(* CODESYS project Simulation_Arm_ROS2_COD_OOP.project

Project tree, tasks and I/O mapping:
  Device : CODESYS Virtual Control for Linux SL, CODESYS, order no. 2302000005, version 4.22.0.0
    application Application
      libraries: Standard, 3.5.22.0 (System); VisuDialogs, * (System)
      task MainTask (cyclic, interval t#20ms, priority 1) calls PLC_PRG, PRG_Visu [Visualisierung]
      program PLC_PRG [ST]
      Kommunikationsverwalter
        OPC UA Server
          Symbolgruppe
      global variables GVL_OPCUA
      visualisation Topics_Vis
      program PRG_VISU [ST]
      Structs/
        ST_RobotStatus/
          data type ST_RobotStatus
          data type ST_Pose_Axis
          data type ST_Pose_TCP
          data type ST_Modes
        ST_RobotAction/
          data type RobotAction
        ST_RobotCommand/
          data type RobotCommand
          data type ST_Servo_Axis
          data type ST_Servo_TCP
      old_code/
        data type Manuell_Achse
        data type TCP_Pose
        data type JointState
        FB_Robot/
          function block FB_Robot [FBD]
          function block FB_Watchdog [ST]
          function block FB_RobotCommand [ST]
      Interfaces/
        interface IF_RobotStatus: Ist_Pose_Axis, Ist_Pose_TCP, Ist_Mode, Client_Connection_Status, Update_Watchdog
        interface IF_RobotCommand: Soll_Pose_Axis, Soll_Pose_TCP
      function block FB_Roboter [FBD]: Update_Watchdog, Soll_Pose_Axis, Soll_Pose_TCP, Client_Connection_Status, Ist_Mode, Ist_Pose_Axis, Ist_Pose_TCP
  libraries: SM3_Robotics, * (CODESYS); VisuSymbols, 4.5.0.0 (System)
  text list GlobalTextList
*)

// Device/Application/old_code/Manuell_Achse
TYPE Manuell_Achse :
STRUCT
	axis_0_plus : BOOL;
	axis_0_minus : BOOL;
	axis_1_plus : BOOL;
	axis_1_minus : BOOL;
	axis_2_plus : BOOL;
	axis_2_minus : BOOL;
	axis_3_plus : BOOL;
	axis_3_minus : BOOL;
	axis_4_plus : BOOL;
	axis_4_minus : BOOL;
	axis_5_plus : BOOL;
	axis_5_minus : BOOL;
	//velocity_spee  einstellen
	//start manuell
END_STRUCT
END_TYPE

// Device/Application/old_code/TCP_Pose
TYPE TCP_Pose :
STRUCT
	trans_x : LREAL;
	trans_y : LREAL;
	trans_z : LREAL;
	rot_x : LREAL;
	rot_y : LREAL;
	rot_z : LREAL;
	rot_w : LREAL;
END_STRUCT
END_TYPE

//TCP Pose in kartesischen Koordinaten
//Rotation wird in quaternions uebermittelt, muss noch umgerechnet werden

// Device/Application/old_code/JointState
TYPE JointState :
STRUCT
	name :ARRAY[0..5] OF STRING;
	position :ARRAY[0..5] OF LREAL; 
	effort :ARRAY[0..5] OF LREAL;
	velocity :ARRAY[0..5] OF LREAL;
END_STRUCT
END_TYPE

// Device/Application/Structs/ST_RobotStatus/ST_RobotStatus
// Gibt den aktuellen Status des Roboters an
TYPE ST_RobotStatus :
STRUCT
	Client_Connected : BOOL;
	Watchdog_Client : INT;		// Überprüft serverseitige client verbindung
	Mode : ST_Modes;			//gibt an ob im Mode Command, Action oder idle
	Pos_Axis : ST_Pose_Axis; 	//gibt aktuelle Achspositionen an
	Pos_TCP : ST_Pose_TCP;		//gibt aktuelle tcp positionen an 
END_STRUCT
END_TYPE

// Device/Application/Structs/ST_RobotCommand/RobotCommand
TYPE RobotCommand :
STRUCT
	Client_connected: BOOL;
	Watchdog_Client: INT;
	axis_servo : ST_Servo_Axis;
	tcp_servo : ST_Servo_TCP;
END_STRUCT
END_TYPE

// Device/Application/Structs/ST_RobotAction/RobotAction
TYPE RobotAction :
STRUCT
END_STRUCT
END_TYPE

// Device/Application/Structs/ST_RobotStatus/ST_Pose_Axis
TYPE ST_Pose_Axis :
STRUCT
	axis_0 : LREAL;
	axis_1 : LREAL;
	axis_2 : LREAL;
	axis_3 : LREAL;
	axis_4 : LREAL;
	axis_5 : LREAL;
END_STRUCT
END_TYPE

// Device/Application/Structs/ST_RobotStatus/ST_Pose_TCP
TYPE ST_Pose_TCP :
STRUCT
	trans_x : LREAL;
	trans_y :  LREAL;
	trans_z : LREAL;
	rot_x : LREAL;
	rot_y : LREAL;
	rot_z : LREAL;
	rot_w : LREAL;
END_STRUCT
END_TYPE

// Device/Application/Structs/ST_RobotStatus/ST_Modes
TYPE ST_Modes :
STRUCT
	idle : BOOL;	//Ruhezustand
	command : BOOL;	//manuell
	aut : BOOL; 	//move_action
END_STRUCT
END_TYPE

// Device/Application/Structs/ST_RobotCommand/ST_Servo_Axis
TYPE ST_Servo_Axis :
STRUCT
	velocity : LREAL;	
	axis_0 : LREAL;
	axis_1 : LREAL;
	axis_2 : LREAL;
	axis_3 : LREAL;
	axis_4 : LREAL;
	axis_5 : LREAL;
END_STRUCT
END_TYPE

// Device/Application/Structs/ST_RobotCommand/ST_Servo_TCP
TYPE ST_Servo_TCP :
STRUCT
	velocity : LREAL;
	trans_x : LREAL;
	trans_y : LREAL;
	trans_z : LREAL;
	rot_x : LREAL;
	rot_y : LREAL;
	rot_z : LREAL;
	rot_w : LREAL;
END_STRUCT
END_TYPE

// Device/Application/GVL_OPCUA
{attribute 'qualified_only'}
VAR_GLOBAL
	PI : REAL := 3.14159;

	//Simulation Arm
	
	//ROS2 -> Codesys
	//topic_name_ros2 : STRUCT
	//joint_states : JointState;	
	//tcp_pose: TCP_Pose;
	
	//achse manuell verfahren
	//axis_manual : Manuell_Achse;
	


END_VAR

// Device/Application/PLC_PRG
PROGRAM PLC_PRG
VAR
END_VAR

END_PROGRAM

// Device/Application/PRG_VISU
PROGRAM PRG_Visu
VAR
    //arrStruct: ARRAY[0..6] OF LREAL;
	Robot : FB_Roboter;
	
END_VAR

Robot();

END_PROGRAM

// Device/Application/FB_Roboter
FUNCTION_BLOCK FB_Roboter IMPLEMENTS IF_RobotCommand, IF_RobotStatus
VAR_INPUT
END_VAR
VAR_OUTPUT
END_VAR
VAR
	// --- Command Variablen ---
    _soll_pose_axis : ST_Servo_Axis; // (Passend zu deinem Struct-Namen)
    _soll_pose_tcp  : ST_Servo_TCP;
    
    // --- Status Variablen ---
    _client_connection_status : BOOL;
    _ist_mode         : ST_Modes;
    _ist_pose_axis    : ST_Pose_Axis;
    _ist_pose_tcp     : ST_Pose_TCP;
END_VAR

// NETWORK 1

{warning 'Methodenimplementierung hinzufügen'}
METHOD Update_Watchdog : BOOL
END_METHOD

{attribute 'monitoring' := 'variable'}
PROPERTY Soll_Pose_Axis : ST_Servo_Axis
GET
END_GET
SET
END_SET
END_PROPERTY

{attribute 'monitoring' := 'variable'}
PROPERTY Soll_Pose_TCP : ST_Servo_TCP
GET
END_GET
SET
END_SET
END_PROPERTY

{attribute 'monitoring' := 'variable'}
PROPERTY Client_Connection_Status : BOOL
GET
Client_Connection_Status := _client_connection_status;
END_GET
SET
_client_connection_status := Client_Connection_Status;
END_SET
END_PROPERTY

{attribute 'monitoring' := 'variable'}
PROPERTY Ist_Mode : ST_Modes
GET
Ist_Mode := _ist_mode;
END_GET
SET
_ist_mode := Ist_Mode;
END_SET
END_PROPERTY

{attribute 'monitoring' := 'variable'}
PROPERTY Ist_Pose_Axis : ST_Pose_Axis
GET
Ist_Pose_Axis := _ist_pose_axis;
END_GET
SET
_ist_pose_axis := Ist_Pose_Axis;
END_SET
END_PROPERTY

{attribute 'monitoring' := 'variable'}
PROPERTY Ist_Pose_TCP : ST_Pose_TCP
GET
Ist_Pose_TCP := _ist_pose_tcp;
END_GET
SET
_ist_pose_tcp := Ist_Pose_TCP;
END_SET
END_PROPERTY

END_FUNCTION_BLOCK

// Device/Application/Interfaces/IF_RobotCommand
INTERFACE IF_RobotCommand

PROPERTY Soll_Pose_Axis : ST_Servo_Axis
SET
END_SET
GET
END_GET
END_PROPERTY

PROPERTY Soll_Pose_TCP : ST_Servo_TCP
SET
END_SET
GET
END_GET
END_PROPERTY

END_INTERFACE

// Device/Application/Interfaces/IF_RobotStatus
INTERFACE IF_RobotStatus

PROPERTY Ist_Pose_Axis : ST_Pose_Axis
GET
END_GET
END_PROPERTY

PROPERTY Ist_Pose_TCP : ST_Pose_TCP
GET
END_GET
END_PROPERTY

PROPERTY Ist_Mode : ST_Modes
SET
END_SET
GET
END_GET
END_PROPERTY

PROPERTY Client_Connection_Status : BOOL
SET
END_SET
GET
END_GET
END_PROPERTY

METHOD Update_Watchdog : BOOL
VAR_INPUT
END_VAR
END_METHOD

END_INTERFACE

// Device/Application/old_code/FB_Robot/FB_Robot
FUNCTION_BLOCK FB_Robot
VAR_INPUT
	Command: RobotCommand;
END_VAR
VAR_OUTPUT
	Status: ST_RobotStatus;
END_VAR
VAR
	robotcommand : FB_RobotCommand;
	Watchdog: FB_Watchdog;
END_VAR

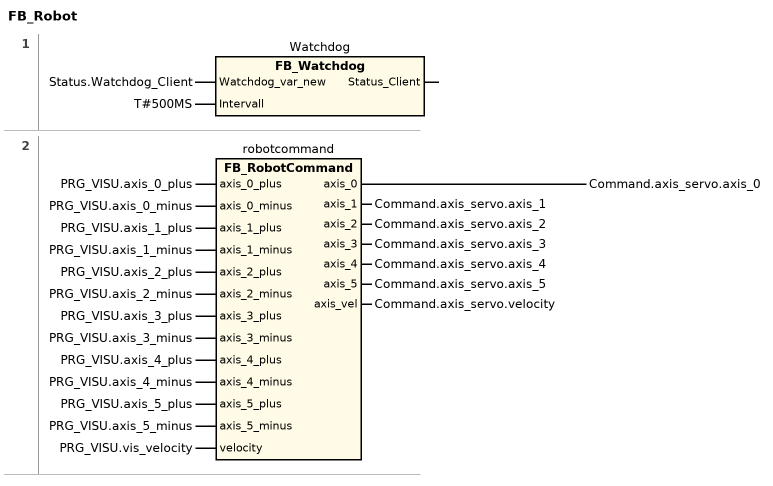
// NETWORK 1
Watchdog(Watchdog_var_new := Status.Watchdog_Client, Intervall := T#500MS); // FB_Watchdog

// NETWORK 2
robotcommand(
    axis_0_plus := PRG_VISU.axis_0_plus,
    axis_0_minus := PRG_VISU.axis_0_minus,
    axis_1_plus := PRG_VISU.axis_1_plus,
    axis_1_minus := PRG_VISU.axis_1_minus,
    axis_2_plus := PRG_VISU.axis_2_plus,
    axis_2_minus := PRG_VISU.axis_2_minus,
    axis_3_plus := PRG_VISU.axis_3_plus,
    axis_3_minus := PRG_VISU.axis_3_minus,
    axis_4_plus := PRG_VISU.axis_4_plus,
    axis_4_minus := PRG_VISU.axis_4_minus,
    axis_5_plus := PRG_VISU.axis_5_plus,
    axis_5_minus := PRG_VISU.axis_5_minus,
    velocity := PRG_VISU.vis_velocity,
    axis_1 => Command.axis_servo.axis_1,
    axis_2 => Command.axis_servo.axis_2,
    axis_3 => Command.axis_servo.axis_3,
    axis_4 => Command.axis_servo.axis_4,
    axis_5 => Command.axis_servo.axis_5,
    axis_vel => Command.axis_servo.velocity); // FB_RobotCommand
Command.axis_servo.axis_0 := robotcommand.axis_0;

END_FUNCTION_BLOCK

// Device/Application/old_code/FB_Robot/FB_Watchdog
FUNCTION_BLOCK FB_Watchdog
VAR_INPUT
	Watchdog_var_new: INT;
	Intervall : TIME;
END_VAR
VAR_OUTPUT
	Status_Client : BOOL;
END_VAR
VAR
	Watchdog_var_old : INT := -1;
	Timer : TON;
END_VAR

IF Watchdog_var_new <> Watchdog_var_old THEN

    Watchdog_var_old := Watchdog_var_new;
    Status_Client := TRUE;
    Timer(IN := FALSE);

ELSE
    Timer(IN := TRUE,PT := Intervall );
END_IF;

IF Timer.Q THEN
    Status_Client := FALSE;
END_IF;

END_FUNCTION_BLOCK

// Device/Application/old_code/FB_Robot/FB_RobotCommand
FUNCTION_BLOCK FB_RobotCommand
VAR_INPUT
	axis_0_plus : BOOL;
	axis_0_minus : BOOL;
	axis_1_plus : BOOL;
	axis_1_minus : BOOL;
	axis_2_plus : BOOL;
	axis_2_minus : BOOL;
	axis_3_plus : BOOL;
	axis_3_minus : BOOL;
	axis_4_plus : BOOL;
	axis_4_minus : BOOL;
	axis_5_plus : BOOL;
	axis_5_minus : BOOL;
	velocity : LREAL;
END_VAR
VAR_OUTPUT
	axis_0 : LREAL;
	axis_1 : LREAL;
	axis_2 : LREAL;
	axis_3 : LREAL;
	axis_4 : LREAL;
	axis_5 : LREAL;
	axis_vel : LREAL;
END_VAR
VAR
END_VAR

// Achse 0
IF axis_0_plus THEN
    axis_0 := 1;
ELSIF axis_0_minus THEN
    axis_0 := -1;
ELSE
    axis_0 := 0;
END_IF;

// Achse 1
IF axis_1_plus THEN
    axis_1 := 1;
ELSIF axis_1_minus THEN
    axis_1 := -1;
ELSE
    axis_1 := 0;
END_IF;

// Achse 2
IF axis_2_plus THEN
    axis_2 := 1;
ELSIF axis_2_minus THEN
    axis_2 := -1;
ELSE
    axis_2 := 0;
END_IF;

// Achse 3
IF axis_3_plus THEN
    axis_3 := 1;
ELSIF axis_3_minus THEN
    axis_3 := -1;
ELSE
    axis_3 := 0;
END_IF;

// Achse 4
IF axis_4_plus THEN
    axis_4 := 1;
ELSIF axis_4_minus THEN
    axis_4 := -1;
ELSE
    axis_4 := 0;
END_IF;

// Achse 5
IF axis_5_plus THEN
    axis_5 := 1;
ELSIF axis_5_minus THEN
    axis_5 := -1;
ELSE
    axis_5 := 0;
END_IF;

// Geschwimdigkeit setzten
axis_vel := velocity;

END_FUNCTION_BLOCK

// Device/Application/Topics_Vis
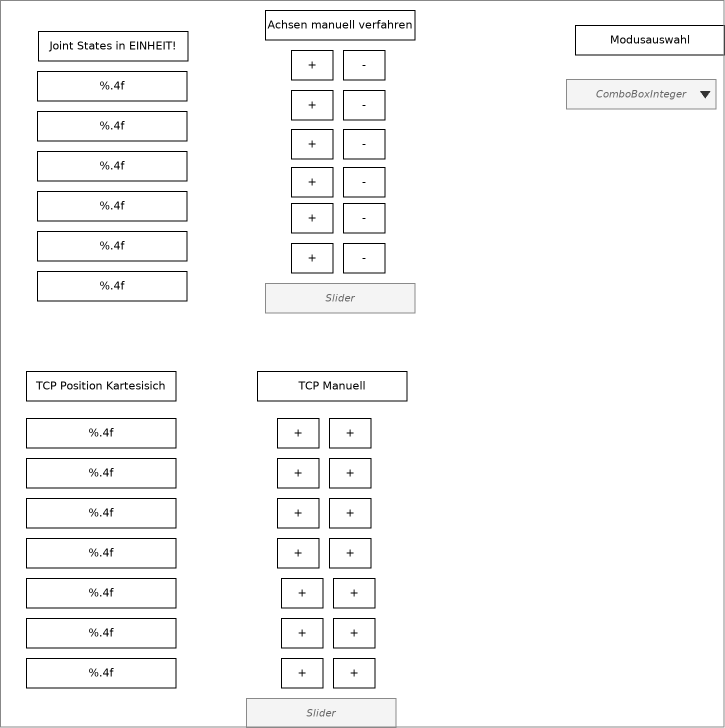
VISUALIZATION Topics_Vis  // 725x728
    Rectangle (38,31 150x30), "Joint States in EINHEIT!"
    Rectangle (26,371 150x30), "TCP Position Kartesisich"
    Rectangle (26,418 150x30), "%.4f", text variable: PRG_Visu.Robot.Status.Pos_TCP.trans_x
    Rectangle (26,458 150x30), "%.4f", text variable: PRG_Visu.Robot.Status.Pos_TCP.trans_y
    Rectangle (26,498 150x30), "%.4f", text variable: PRG_Visu.Robot.Status.Pos_TCP.trans_z
    Rectangle (26,538 150x30), "%.4f", text variable: PRG_Visu.Robot.Status.Pos_TCP.rot_x
    Rectangle (26,578 150x30), "%.4f", text variable: PRG_Visu.Robot.Status.Pos_TCP.rot_y
    Rectangle (26,618 150x30), "%.4f", text variable: PRG_Visu.Robot.Status.Pos_TCP.rot_z
    Rectangle (26,658 150x30), "%.4f", text variable: PRG_Visu.Robot.Status.Pos_TCP.rot_w
    Rectangle (291,50 42x30), "+"
        toggle PRG_Visu.axis_0_plus
    Rectangle (343,50 42x30), "-"
        tap PRG_Visu.axis_0_minus
    Rectangle (291,90 42x30), "+"
        toggle PRG_Visu.axis_1_plus
    Rectangle (343,129 42x30), "-"
    Rectangle (291,129 42x30), "+"
    Rectangle (291,167 42x30), "+"
    Rectangle (343,90 42x30), "-"
        toggle PRG_Visu.axis_1_minus
    Rectangle (343,167 42x30), "-"
    Rectangle (291,203 42x30), "+"
    Rectangle (343,203 42x30), "-"
    Rectangle (291,243 42x30), "+"
    Rectangle (343,243 42x30), "-"
    Slider (265,283 150x30), scale 0..100
    Rectangle (575,25 150x30), "Modusauswahl"
    ComboBoxInteger (566,79 150x30)
    Rectangle (37,71 150x30), "%.4f", text variable: PRG_Visu.Robot.Status.Pos_Axis.axis_0
    Rectangle (37,111 150x30), "%.4f", text variable: PRG_Visu.Robot.Status.Pos_Axis.axis_1
    Rectangle (37,151 150x30), "%.4f", text variable: PRG_Visu.Robot.Status.Pos_Axis.axis_2
    Rectangle (37,191 150x30), "%.4f", text variable: PRG_Visu.Robot.Status.Pos_Axis.axis_3
    Rectangle (37,231 150x30), "%.4f", text variable: PRG_Visu.Robot.Status.Pos_Axis.axis_4
    Rectangle (37,271 150x30), "%.4f", text variable: PRG_Visu.Robot.Status.Pos_Axis.axis_5
    Rectangle (277,418 42x30), "+"
    Rectangle (277,458 42x30), "+"
    Rectangle (277,498 42x30), "+"
    Rectangle (277,538 42x30), "+"
    Rectangle (281,578 42x30), "+"
    Rectangle (281,618 42x30), "+"
    Rectangle (281,658 42x30), "+"
    Rectangle (329,418 42x30), "+"
    Rectangle (329,458 42x30), "+"
    Rectangle (329,498 42x30), "+"
    Rectangle (329,538 42x30), "+"
    Rectangle (333,578 42x30), "+"
    Rectangle (333,618 42x30), "+"
    Rectangle (333,658 42x30), "+"
    Slider (246,698 150x30), scale 0..100
    Rectangle (257,371 150x30), "TCP Manuell"
    Rectangle (265,10 150x30), "Achsen manuell verfahren"
END_VISUALIZATION
